{attribute 'OPC.UA.DA.StructuredType' := '1'}
{attribute 'OPC.UA.DA' := '1'}
TYPE stVisStatusManip :
STRUCT
	State:  eState;
	Mode: eMode;
	isMoving: BOOL;
	isReady: BOOL;
	isConnected: BOOL;
// 	isLocked: BOOL;
	isBusy: BOOL;
	isInCollision: BOOL;
	hasError: BOOL;
	TCPPosition: stPose3D;
END_STRUCT
END_TYPE

(* stored: Version 1.1.0.1, ProductVersion 3.1.4026.18
   DUT stVisStatusManip: Id {49a014e9-2e0d-496e-a201-ae51c8ca9573} *)
